KUKA KRL program: chk_w7_wechs_ok.src

&ACCESS RV6
&COMMENT Check Gripper Axor
DEF chk_w7_wechs_ok( )

; VERIFICAÇÃO DE FERRAMENTA: Gripper Axor

$TIMER[10] = 0
$TIMER_STOP[10] = FALSE

wait for (($in[161]) and ($in[169]) and ($in[177]) and ($IN[185]) and ($IN[193]) and ($IN[201]) and (not $IN[209]) and ($IN[219]))

$TIMER_STOP[10] = TRUE
$TIMER[10] = 0

;//---- End -------
;Diag_Appl(#Off,5)

END
